      A     #i_CMD_Reset;
      O     #t_Suppress_Errors;
      O     #t_Suppress_Errors_Isafe;
      R     #s_Status.SafetyRelais_Err_GRP01;
      R     #s_Status.SafetyRelais_Err_GRP02;
      R     #s_Status.SafetyRelais_Err_GRP03;
      R     #s_Status.SafetyRelais_Err_GRP04;
      R     #s_Status.SafetyRelais_Err_GRP05;
      R     #s_Status.SafetyRelais_Err_GRP06;
      R     #s_Status.SafetyRelais_Err_GRP07;
      R     #s_Status.SafetyRelais_Err_GRP08;
      R     #s_Status.SafetyRelais_Err_GRP09;
      R     #s_Status.SafetyRelais_Err_GRP10;
      R     #s_Status.SafetyRelais_Err_GRP11;
      R     #s_Status.SafetyRelais_Err_GRP12;
      R     #s_Status.SafetyRelais_Err_GRP13;
      R     #s_Status.SafetyRelais_Err_GRP14;
      R     #s_Status.SafetyRelais_Err_GRP15;
      R     #s_Status.SafetyRelais_Err_GRP16;

//Feedback Safety Relay Group 1 Alarm
      A     #i_CFG_Isafe_Used;
      A     #i_SafetyRelais_Err_GRP01;
      S     #s_Status.SafetyRelais_Err_GRP01;

//Feedback Safety Relay Group 2 Alarm
      A     #i_CFG_Isafe_Used;
      A     #i_SafetyRelais_Err_GRP02;
      S     #s_Status.SafetyRelais_Err_GRP02;

//Feedback Safety Relay Group 3 Alarm
      A     #i_CFG_Isafe_Used;
      A     #i_SafetyRelais_Err_GRP03;
      S     #s_Status.SafetyRelais_Err_GRP03;

//Feedback Safety Relay Group 4 Alarm
      A     #i_CFG_Isafe_Used;
      A     #i_SafetyRelais_Err_GRP04;
      S     #s_Status.SafetyRelais_Err_GRP04;

//Feedback Safety Relay Group 5 Alarm
      A     #i_CFG_Isafe_Used;
      A     #i_SafetyRelais_Err_GRP05;
      S     #s_Status.SafetyRelais_Err_GRP05;

//Feedback Safety Relay Group 6 Alarm
      A     #i_CFG_Isafe_Used;
      A     #i_SafetyRelais_Err_GRP06;
      S     #s_Status.SafetyRelais_Err_GRP06;

//Feedback Safety Relay Group 7 Alarm
      A     #i_CFG_Isafe_Used;
      A     #i_SafetyRelais_Err_GRP07;
      S     #s_Status.SafetyRelais_Err_GRP07;

//Feedback Safety Relay Group 8 Alarm
      A     #i_CFG_Isafe_Used;
      A     #i_SafetyRelais_Err_GRP08;
      S     #s_Status.SafetyRelais_Err_GRP08;

//Feedback Safety Relay Group 9 Alarm
      A     #i_CFG_Isafe_Used;
      A     #i_SafetyRelais_Err_GRP09;
      S     #s_Status.SafetyRelais_Err_GRP09;

//Feedback Safety Relay Group 10 Alarm
      A     #i_CFG_Isafe_Used;
      A     #i_SafetyRelais_Err_GRP10;
      S     #s_Status.SafetyRelais_Err_GRP10;

//Feedback Safety Relay Group 11 Alarm
      A     #i_CFG_Isafe_Used;
      A     #i_SafetyRelais_Err_GRP11;
      S     #s_Status.SafetyRelais_Err_GRP11;

//Feedback Safety Relay Group 12 Alarm
      A     #i_CFG_Isafe_Used;
      A     #i_SafetyRelais_Err_GRP12;
      S     #s_Status.SafetyRelais_Err_GRP12;

//Feedback Safety Relay Group 13 Alarm
      A     #i_CFG_Isafe_Used;
      A     #i_SafetyRelais_Err_GRP13;
      S     #s_Status.SafetyRelais_Err_GRP13;

//Feedback Safety Relay Group 14 Alarm
      A     #i_CFG_Isafe_Used;
      A     #i_SafetyRelais_Err_GRP14;
      S     #s_Status.SafetyRelais_Err_GRP14;

//Feedback Safety Relay Group 15 Alarm
      A     #i_CFG_Isafe_Used;
      A     #i_SafetyRelais_Err_GRP15;
      S     #s_Status.SafetyRelais_Err_GRP15;

//Feedback Safety Relay Group 16 Alarm
      A     #i_CFG_Isafe_Used;
      A     #i_SafetyRelais_Err_GRP16;
      S     #s_Status.SafetyRelais_Err_GRP16;



//Mapping Status bit to Output Bit

      A     #s_Status.SafetyRelais_Err_GRP01;
      =     #o_SafetyRelais_Err_GRP01;

      A     #s_Status.SafetyRelais_Err_GRP02;
      =     #o_SafetyRelais_Err_GRP02;

      A     #s_Status.SafetyRelais_Err_GRP03;
      =     #o_SafetyRelais_Err_GRP03;

      A     #s_Status.SafetyRelais_Err_GRP04;
      =     #o_SafetyRelais_Err_GRP04;

      A     #s_Status.SafetyRelais_Err_GRP05;
      =     #o_SafetyRelais_Err_GRP05;

      A     #s_Status.SafetyRelais_Err_GRP06;
      =     #o_SafetyRelais_Err_GRP06;

      A     #s_Status.SafetyRelais_Err_GRP07;
      =     #o_SafetyRelais_Err_GRP07;

      A     #s_Status.SafetyRelais_Err_GRP08;
      =     #o_SafetyRelais_Err_GRP08;

      A     #s_Status.SafetyRelais_Err_GRP09;
      =     #o_SafetyRelais_Err_GRP09;

      A     #s_Status.SafetyRelais_Err_GRP10;
      =     #o_SafetyRelais_Err_GRP10;

      A     #s_Status.SafetyRelais_Err_GRP11;
      =     #o_SafetyRelais_Err_GRP11;


      A     #s_Status.SafetyRelais_Err_GRP12;
      =     #o_SafetyRelais_Err_GRP12;

      A     #s_Status.SafetyRelais_Err_GRP13;
      =     #o_SafetyRelais_Err_GRP13;

      A     #s_Status.SafetyRelais_Err_GRP14;
      =     #o_SafetyRelais_Err_GRP14;

      A     #s_Status.SafetyRelais_Err_GRP15;
      =     #o_SafetyRelais_Err_GRP15;

      A     #s_Status.SafetyRelais_Err_GRP16;
      =     #o_SafetyRelais_Err_GRP16;

NETWORK
TITLE =JA: Safety Signal Handling
//Handle safety stop signals for every motor group
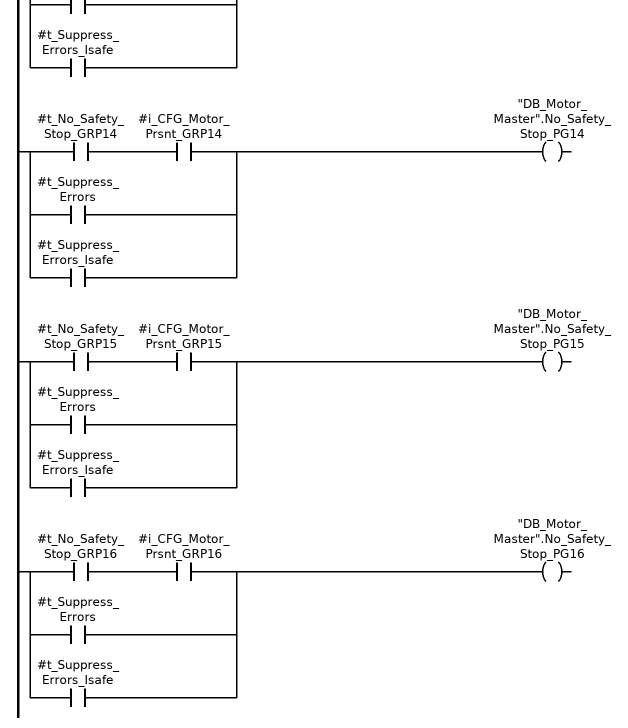
      NOP   0;
// No Safety stop MotorGroup 1
      A     #t_No_Safety_Stop_GRP01;
      A     #i_CFG_Motor_Prsnt_GRP01;
      O     #t_Suppress_Errors;
      O     #t_Suppress_Errors_Isafe;
      =     "DB_Motor_Master".No_Safety_Stop_PG01;

// No Safety stop MotorGroup 2
      A     #t_No_Safety_Stop_GRP02;
      A     #i_CFG_Motor_Prsnt_GRP02;
      O     #t_Suppress_Errors;
      O     #t_Suppress_Errors_Isafe;
      =     "DB_Motor_Master".No_Safety_Stop_PG02;

// No Safety stop MotorGroup 3
      A     #t_No_Safety_Stop_GRP03;
      A     #i_CFG_Motor_Prsnt_GRP03;
      O     #t_Suppress_Errors;
      O     #t_Suppress_Errors_Isafe;
      =     "DB_Motor_Master".No_Safety_Stop_PG03;

// No Safety stop MotorGroup 4
      A     #t_No_Safety_Stop_GRP04;
      A     #i_CFG_Motor_Prsnt_GRP04;
      O     #t_Suppress_Errors;
      O     #t_Suppress_Errors_Isafe;
      =     "DB_Motor_Master".No_Safety_Stop_PG04;

// No Safety stop MotorGroup 5
      A     #t_No_Safety_Stop_GRP05;
      A     #i_CFG_Motor_Prsnt_GRP05;
      O     #t_Suppress_Errors;
      O     #t_Suppress_Errors_Isafe;
      =     "DB_Motor_Master".No_Safety_Stop_PG05;

// No Safety stop MotorGroup 6
      A     #t_No_Safety_Stop_GRP06;
      A     #i_CFG_Motor_Prsnt_GRP06;
      O     #t_Suppress_Errors;
      O     #t_Suppress_Errors_Isafe;
      =     "DB_Motor_Master".No_Safety_Stop_PG06;

// No Safety stop MotorGroup 7
      A     #t_No_Safety_Stop_GRP07;
      A     #i_CFG_Motor_Prsnt_GRP07;
      O     #t_Suppress_Errors;
      O     #t_Suppress_Errors_Isafe;
      =     "DB_Motor_Master".No_Safety_Stop_PG07;

// No Safety stop MotorGroup 8
      A     #t_No_Safety_Stop_GRP08;
      A     #i_CFG_Motor_Prsnt_GRP08;
      O     #t_Suppress_Errors;
      O     #t_Suppress_Errors_Isafe;
      =     "DB_Motor_Master".No_Safety_Stop_PG08;

// No Safety stop MotorGroup 9
      A     #t_No_Safety_Stop_GRP09;
      A     #i_CFG_Motor_Prsnt_GRP09;
      O     #t_Suppress_Errors;
      O     #t_Suppress_Errors_Isafe;
      =     "DB_Motor_Master".No_Safety_Stop_PG09;

// No Safety stop MotorGroup 10
      A     #t_No_Safety_Stop_GRP10;
      A     #i_CFG_Motor_Prsnt_GRP10;
      O     #t_Suppress_Errors;
      O     #t_Suppress_Errors_Isafe;
      =     "DB_Motor_Master".No_Safety_Stop_PG10;

// No Safety stop MotorGroup 11
      A     #t_No_Safety_Stop_GRP11;
      A     #i_CFG_Motor_Prsnt_GRP11;
      O     #t_Suppress_Errors;
      O     #t_Suppress_Errors_Isafe;
      =     "DB_Motor_Master".No_Safety_Stop_PG11;

// No Safety stop MotorGroup 12
      A     #t_No_Safety_Stop_GRP12;
      A     #i_CFG_Motor_Prsnt_GRP12;
      O     #t_Suppress_Errors;
      O     #t_Suppress_Errors_Isafe;
      =     "DB_Motor_Master".No_Safety_Stop_PG12;

// No Safety stop MotorGroup 13
      A     #t_No_Safety_Stop_GRP13;
      A     #i_CFG_Motor_Prsnt_GRP13;
      O     #t_Suppress_Errors;
      O     #t_Suppress_Errors_Isafe;
      =     "DB_Motor_Master".No_Safety_Stop_PG13;

// No Safety stop MotorGroup 14
      A     #t_No_Safety_Stop_GRP14;
      A     #i_CFG_Motor_Prsnt_GRP14;
      O     #t_Suppress_Errors;
      O     #t_Suppress_Errors_Isafe;
      =     "DB_Motor_Master".No_Safety_Stop_PG14;

// No Safety stop MotorGroup 15
      A     #t_No_Safety_Stop_GRP15;
      A     #i_CFG_Motor_Prsnt_GRP15;
      O     #t_Suppress_Errors;
      O     #t_Suppress_Errors_Isafe;
      =     "DB_Motor_Master".No_Safety_Stop_PG15;

// No Safety stop MotorGroup 16
      A     #t_No_Safety_Stop_GRP16;
      A     #i_CFG_Motor_Prsnt_GRP16;
      O     #t_Suppress_Errors;
      O     #t_Suppress_Errors_Isafe;
      =     "DB_Motor_Master".No_Safety_Stop_PG16;

NETWORK
TITLE =KA: Handle commands
//Set the controlled stop and direct stop output signals.
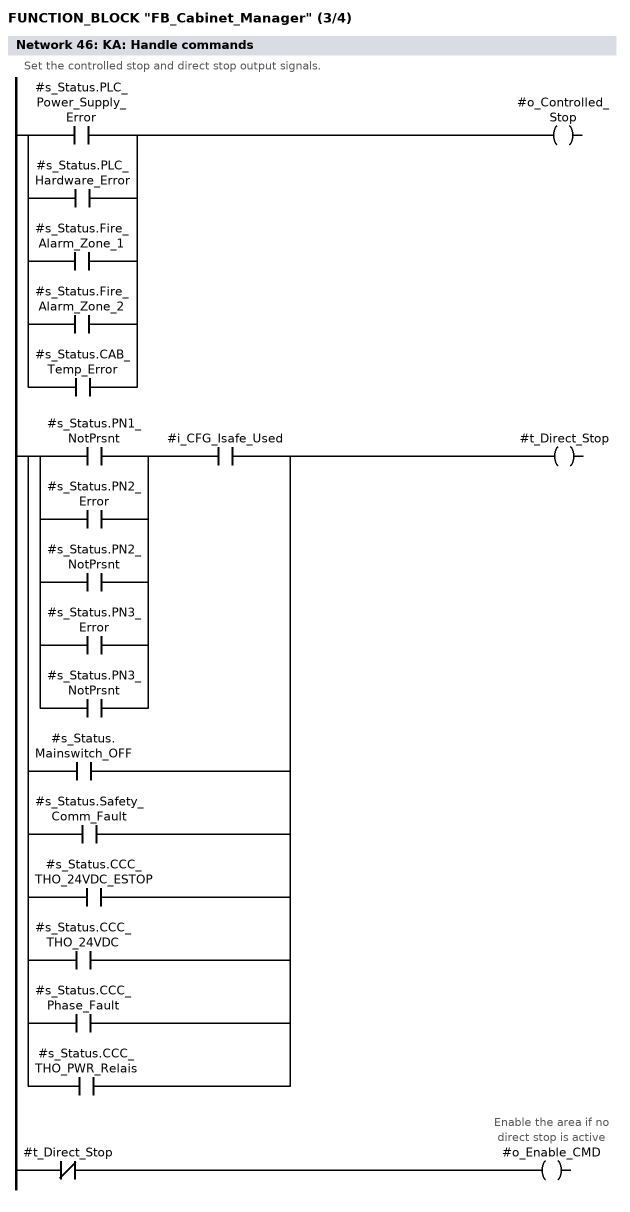
      O     #s_Status.PLC_Power_Supply_Error;
      O     #s_Status.PLC_Hardware_Error;
      O     #s_Status.Fire_Alarm_Zone_1;
      O     #s_Status.Fire_Alarm_Zone_2;
      O     #s_Status.CAB_Temp_Error;
      =     #o_Controlled_Stop;

      A(    ;
      O     #s_Status.PN1_NotPrsnt;
      O     #s_Status.PN2_Error;
      O     #s_Status.PN2_NotPrsnt;
      O     #s_Status.PN3_Error;
      O     #s_Status.PN3_NotPrsnt;
      )     ;
      A     #i_CFG_Isafe_Used;
      O     #s_Status.Mainswitch_OFF;
      O     #s_Status.Safety_Comm_Fault;
      O     #s_Status.CCC_THO_24VDC_ESTOP;
      O     #s_Status.CCC_THO_24VDC;
// Option to stop is Phase fault is detected.
      O     #s_Status.CCC_Phase_Fault;
      O     #s_Status.CCC_THO_PWR_Relais;
      =     #t_Direct_Stop;

      AN    #t_Direct_Stop;
      =     #o_Enable_CMD; //Enable the area if no direct stop is active
NETWORK
TITLE =LA: Write output signals
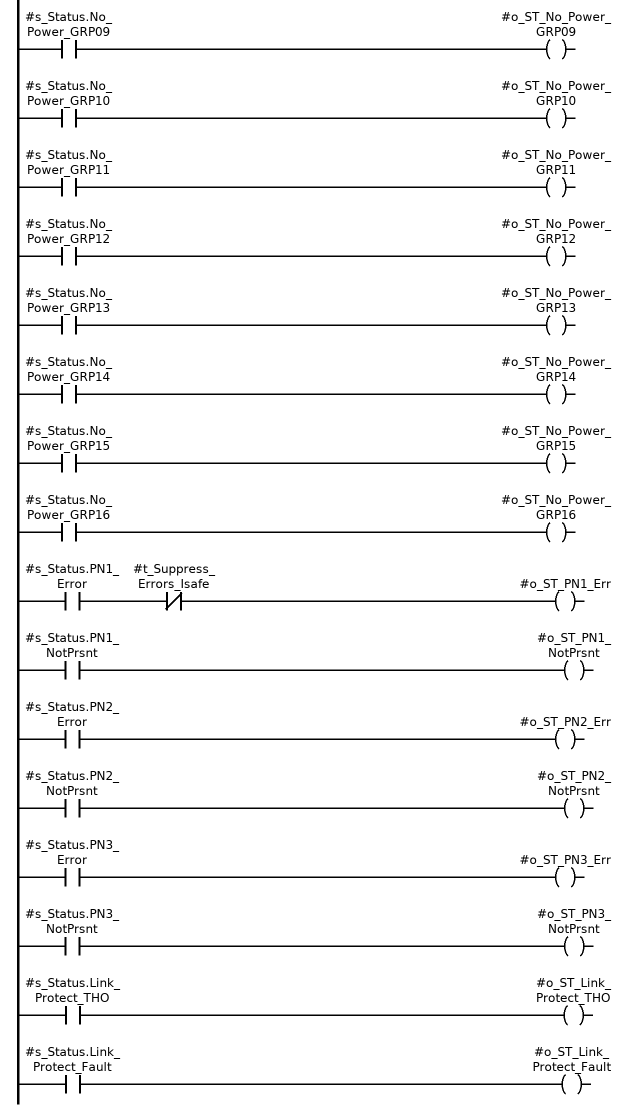

      A     #s_Status.Mainswitch_OFF;
      =     #o_ST_Mainswitch_OFF;

      A     #s_Status.PLC_Power_Supply_Error;
      =     #o_ST_PLC_Power_Supply_Er;

      A     #s_Status.PLC_Hardware_Error;
      =     #o_ST_PLC_Hardware_Er;

      A     #s_Status.PLC_Battery_Error;
      =     #o_ST_PLC_Battery_Er;

      A     #s_Status.Safety_Comm_Fault;
      AN    #t_Suppress_Errors_Isafe;
      =     #o_ST_Safety_Comm_Fault;

      A     #s_Status.CCC_THO_24VDC;
      =     #o_ST_CCC_THO_24VDC;

      A     #s_Status.CCC_THO_24VDC_ESTOP;
      =     #o_ST_CCC_THO_24VDC_ESTOP;

      A     #s_Status.CCC_THO_AMP;
      =     #o_ST_CCC_THO_AMP;

      A     #s_Status.CCC_THO_Phase;
      =     #o_ST_CCC_THO_Phase;

      A     #s_Status.CCC_Phase_Fault;
      =     #o_ST_CCC_Phase_Fault;

      A     #s_Status.CCC_THO_PWR_Relais;
      =     #o_ST_CCC_THO_PWR_Relais;

      A     #s_Status.Fire_Alarm_Zone_1;
      =     #o_ST_Fire_Alarm_Zone_1;

      A     #s_Status.Fire_Alarm_Zone_2;
      =     #o_ST_Fire_Alarm_Zone_2;

      A     #s_Status.ETH_Switch_Fault;
      =     #o_ST_ETH_Switch_Fault;

      A     #s_Status.CAB_Temp_High;
      =     #o_ST_CAB_Temp_High;

      A     #s_Status.CAB_Temp_Error;
      =     #o_ST_CAB_Temp_Error;

      A     #s_Status.UPS_THO;
      =     #o_ST_UPS_THO;

      A     #s_Status.PN_Master_Error;
      =     #o_ST_PN_Mstr_Err;

      A     #s_Status.PN_Master_NotPrsnt;
      =     #o_ST_PN_Mstr_NotPrsnt;

      A     #s_Status.THO_Main_Pwr_GRP01;
      =     #o_ST_THO_Main_Pwr_GRP01;

      A     #s_Status.THO_Main_Pwr_GRP02;
      =     #o_ST_THO_Main_Pwr_GRP02;

      A     #s_Status.THO_Main_Pwr_GRP03;
      =     #o_ST_THO_Main_Pwr_GRP03;

      A     #s_Status.THO_Main_Pwr_GRP04;
      =     #o_ST_THO_Main_Pwr_GRP04;

      A     #s_Status.THO_Main_Pwr_GRP05;
      =     #o_ST_THO_Main_Pwr_GRP05;

      A     #s_Status.THO_Main_Pwr_GRP06;
      =     #o_ST_THO_Main_Pwr_GRP06;

      A     #s_Status.THO_Main_Pwr_GRP07;
      =     #o_ST_THO_Main_Pwr_GRP07;

      A     #s_Status.THO_Main_Pwr_GRP08;
      =     #o_ST_THO_Main_Pwr_GRP08;

      A     #s_Status.THO_Main_Pwr_GRP09;
      =     #o_ST_THO_Main_Pwr_GRP09;

      A     #s_Status.THO_Main_Pwr_GRP10;
      =     #o_ST_THO_Main_Pwr_GRP10;

      A     #s_Status.THO_Main_Pwr_GRP11;
      =     #o_ST_THO_Main_Pwr_GRP11;

      A     #s_Status.THO_Main_Pwr_GRP12;
      =     #o_ST_THO_Main_Pwr_GRP12;

      A     #s_Status.THO_Main_Pwr_GRP13;
      =     #o_ST_THO_Main_Pwr_GRP13;

      A     #s_Status.THO_Main_Pwr_GRP14;
      =     #o_ST_THO_Main_Pwr_GRP14;

      A     #s_Status.THO_Main_Pwr_GRP15;
      =     #o_ST_THO_Main_Pwr_GRP15;

      A     #s_Status.THO_Main_Pwr_GRP16;
      =     #o_ST_THO_Main_Pwr_GRP16;

      A     #s_Status.THO_Aux_Pwr_GRP01;
      =     #o_ST_THO_Aux_Pwr_GRP01;

      A     #s_Status.THO_Aux_Pwr_GRP02;
      =     #o_ST_THO_Aux_Pwr_GRP02;

      A     #s_Status.THO_Aux_Pwr_GRP03;
      =     #o_ST_THO_Aux_Pwr_GRP03;

      A     #s_Status.THO_Aux_Pwr_GRP04;
      =     #o_ST_THO_Aux_Pwr_GRP04;

      A     #s_Status.THO_Aux_Pwr_GRP05;
      =     #o_ST_THO_Aux_Pwr_GRP05;

      A     #s_Status.THO_Aux_Pwr_GRP06;
      =     #o_ST_THO_Aux_Pwr_GRP06;

      A     #s_Status.THO_Aux_Pwr_GRP07;
      =     #o_ST_THO_Aux_Pwr_GRP07;

      A     #s_Status.THO_Aux_Pwr_GRP08;
      =     #o_ST_THO_Aux_Pwr_GRP08;

      A     #s_Status.THO_Aux_Pwr_GRP09;
      =     #o_ST_THO_Aux_Pwr_GRP09;

      A     #s_Status.THO_Aux_Pwr_GRP10;
      =     #o_ST_THO_Aux_Pwr_GRP10;

      A     #s_Status.THO_Aux_Pwr_GRP11;
      =     #o_ST_THO_Aux_Pwr_GRP11;

      A     #s_Status.THO_Aux_Pwr_GRP12;
      =     #o_ST_THO_Aux_Pwr_GRP12;

      A     #s_Status.THO_Aux_Pwr_GRP13;
      =     #o_ST_THO_Aux_Pwr_GRP13;

      A     #s_Status.THO_Aux_Pwr_GRP14;
      =     #o_ST_THO_Aux_Pwr_GRP14;

      A     #s_Status.THO_Aux_Pwr_GRP15;
      =     #o_ST_THO_Aux_Pwr_GRP15;

      A     #s_Status.THO_Aux_Pwr_GRP16;
      =     #o_ST_THO_Aux_Pwr_GRP16;

      A     #s_Status.No_Power_GRP01;
      =     #o_ST_No_Power_GRP01;

      A     #s_Status.No_Power_GRP02;
      =     #o_ST_No_Power_GRP02;

      A     #s_Status.No_Power_GRP03;
      =     #o_ST_No_Power_GRP03;

      A     #s_Status.No_Power_GRP04;
      =     #o_ST_No_Power_GRP04;

      A     #s_Status.No_Power_GRP05;
      =     #o_ST_No_Power_GRP05;

      A     #s_Status.No_Power_GRP06;
      =     #o_ST_No_Power_GRP06;

      A     #s_Status.No_Power_GRP07;
      =     #o_ST_No_Power_GRP07;

      A     #s_Status.No_Power_GRP08;
      =     #o_ST_No_Power_GRP08;

      A     #s_Status.No_Power_GRP09;
      =     #o_ST_No_Power_GRP09;

      A     #s_Status.No_Power_GRP10;
      =     #o_ST_No_Power_GRP10;

      A     #s_Status.No_Power_GRP11;
      =     #o_ST_No_Power_GRP11;

      A     #s_Status.No_Power_GRP12;
      =     #o_ST_No_Power_GRP12;

      A     #s_Status.No_Power_GRP13;
      =     #o_ST_No_Power_GRP13;

      A     #s_Status.No_Power_GRP14;
      =     #o_ST_No_Power_GRP14;

      A     #s_Status.No_Power_GRP15;
      =     #o_ST_No_Power_GRP15;

      A     #s_Status.No_Power_GRP16;
      =     #o_ST_No_Power_GRP16;

      A     #s_Status.PN1_Error;
      AN    #t_Suppress_Errors_Isafe;
      =     #o_ST_PN1_Err;

      A     #s_Status.PN1_NotPrsnt;
      =     #o_ST_PN1_NotPrsnt;

      A     #s_Status.PN2_Error;
      =     #o_ST_PN2_Err;

      A     #s_Status.PN2_NotPrsnt;
      =     #o_ST_PN2_NotPrsnt;

      A     #s_Status.PN3_Error;
      =     #o_ST_PN3_Err;

      A     #s_Status.PN3_NotPrsnt;
      =     #o_ST_PN3_NotPrsnt;

      A     #s_Status.Link_Protect_THO;
      =     #o_ST_Link_Protect_THO;

      A     #s_Status.Link_Protect_Fault;
      =     #o_ST_Link_Protect_Fault;
END_FUNCTION_BLOCK

